ABB RobotStudio station: Solution_1.rspag

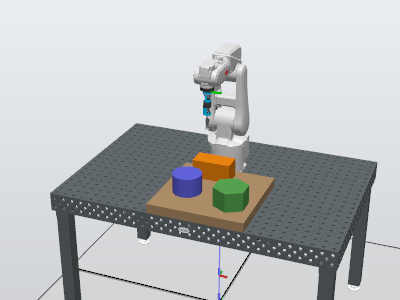
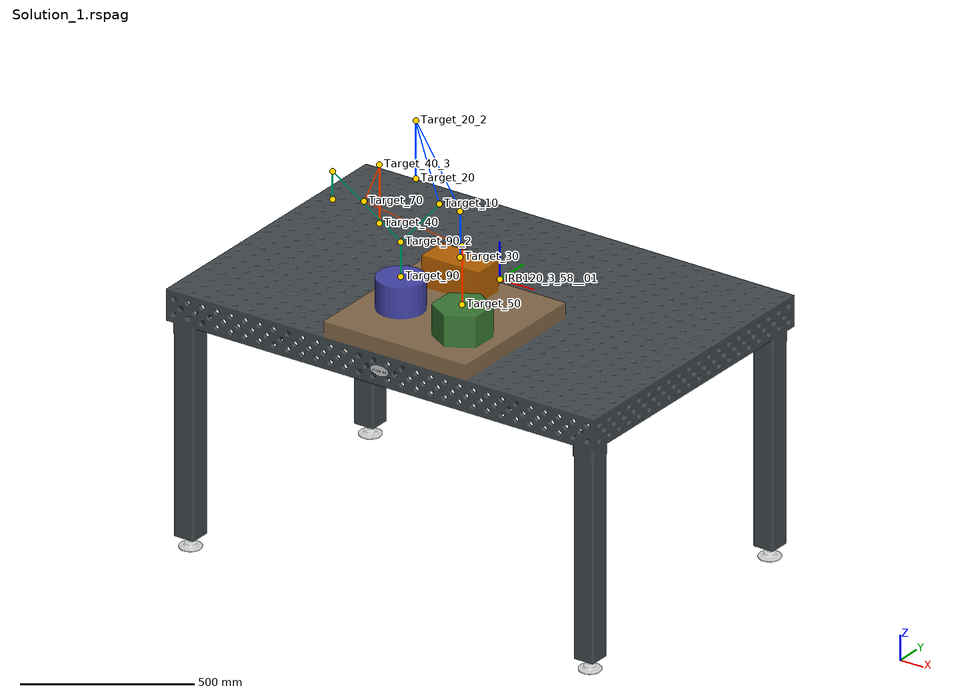
[picture v1: parts stored in the station drawn from their meshes, with robot base, taught points and paths (robot models come from the ABB library and are not in the file)]
--- station ---
Station Solution_1_Tutorial (saved by RobotStudio 22.3.10190.2)
Controller Controller1, task T_ROB1: task frame (RAPID world) sits at (0, 100, 830) mm, rotated rx 0 ry 0 rz -90 deg in the station
Controller Controller1
  mechanical unit ROB_1: IRB120_3_58__01, 6 joints, base frame (0, 0, 0) mm
Layout (positions relative to the parent item):
  - table [part] at (-200, -500, 830) mm, size 500 x 500 x 50 mm
  - object_1 [part] at (-200, -500, 830) mm, size 200 x 100 x 150 mm
  - object_2 [part] at (-200, -500, 830) mm, size 149.5 x 149.7 x 150 mm
  - object_3 [part] at (-200, -500, 830) mm, size 155.5 x 179.5 x 150 mm
  - siegmund_1500_1000 [part], size 1500 x 1010.3 x 830 mm
  - object_11 [part] at (-200, -500, 830) mm, size 200 x 100 x 150 mm
  - object_22 [part] at (-200, -500, 830) mm, size 149.5 x 149.7 x 150 mm
  - object_33 [part] at (-200, -500, 830) mm, size 155.5 x 179.5 x 150 mm
  - IRB120_3_58__01 [mechanism, from Robots\IRB120_3_58_G_01.rslib] at (0, 100, 830) mm, rotated rx 0 ry 0 rz -90 deg; joint values [0, 0, 0, 0, 1.5708, 0] (rad or m)
  - smc_gripper [mechanism, from Gripper_RS_tool\smc_gripper.rslib] at (0, -202, 1388) mm, rotated rx 180 ry 0 rz 90 deg
  - Attacher [smart component, from Components\Attacher.rslib]
      properties: Parent=smc_gripper; Flange=0; Child=object_1; Mount=false; Offset=[0 0 0]; Orientation=[0 0 0]
  - Detacher [smart component, from Components\Detacher.rslib]
      properties: Child=object_1; KeepPosition=true
  - Positioner [smart component, from Components\Positioner.rslib] at (-600, -150, 830) mm
      properties: Object=object_1; Position=[-0.6 -0.15 0.83]; Orientation=[0 0 0]; Reference=Global; ReferenceObject=(none)
  - Detacher_2 [smart component, from Components\Detacher.rslib]
      properties: Child=object_3; KeepPosition=true
  - Attacher_2 [smart component, from Components\Attacher.rslib]
      properties: Parent=smc_gripper; Flange=0; Child=object_3; Mount=false; Offset=[0 0 0]; Orientation=[0 0 0]
  - Attacher_3 [smart component, from Components\Attacher.rslib]
      properties: Parent=smc_gripper; Flange=0; Child=object_2; Mount=false; Offset=[0 0 0]; Orientation=[0 0 0]
  - Detacher_3 [smart component, from Components\Detacher.rslib]
      properties: Child=object_2; KeepPosition=true
  - Positioner_2 [smart component, from Components\Positioner.rslib]
      properties: Object=object_3; Position=[-0.7 -0.2 0.83]; Orientation=[0 0 0]; Reference=Global; ReferenceObject=(none)
  - Positioner_3 [smart component, from Components\Positioner.rslib]
      properties: Object=object_2; Position=[-0.65 -0.2 0.83]; Orientation=[0 0 0]; Reference=Global; ReferenceObject=(none)
  - Frame_1 [frame] at (0, 0, 197) mm
Attachment: smc_gripper is attached to IRB120_3_58__01 / Link6
Station signals: DI DI_TEST_01
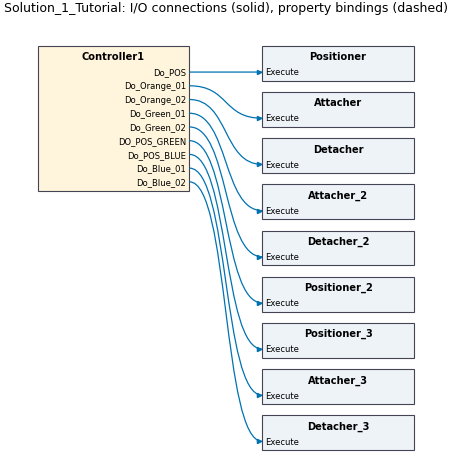
Station logic (signal -> signal, property => property):
  Controller1.Do_POS -> Positioner.Execute
  Controller1.Do_Orange_01 -> Attacher.Execute
  Controller1.Do_Orange_02 -> Detacher.Execute
  Controller1.Do_Green_01 -> Attacher_2.Execute
  Controller1.Do_Green_02 -> Detacher_2.Execute
  Controller1.DO_POS_GREEN -> Positioner_2.Execute
  Controller1.Do_POS_BLUE -> Positioner_3.Execute
  Controller1.Do_Blue_01 -> Attacher_3.Execute
  Controller1.Do_Blue_02 -> Detacher_3.Execute

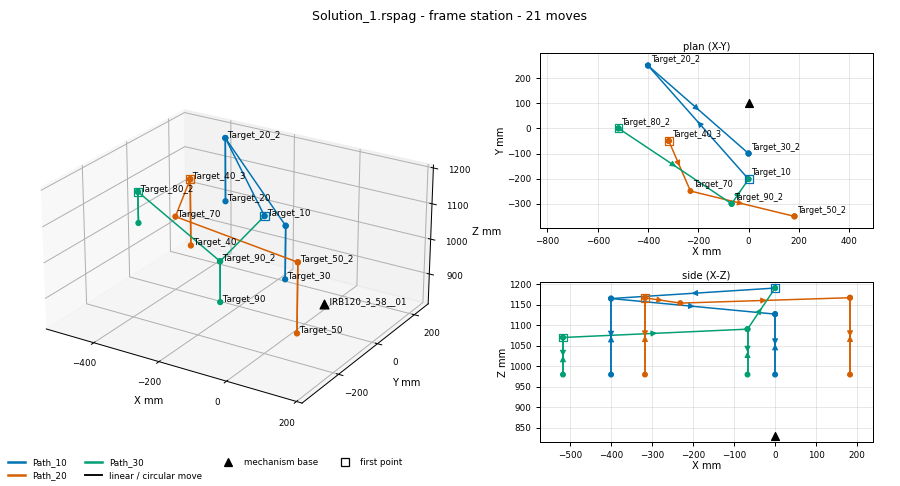
[picture p0: tool path of Solution_1.rspag in frame station, 21 of 21 moves have a stored position in this frame; points joined in program order, loops and branches not executed]
--- Backups/Controller1/RAPID/TASK1/PROGMOD/CalibData.mod ---
MODULE CalibData
    PERS tooldata smc_gripper:=[TRUE,[[0,0.004,197.001],[1,0,0,0]],[1,[0.207,-0.496,71.18],[1,0,0,0],0,0,0]];
ENDMODULE

--- Backups/Controller1/RAPID/TASK1/PROGMOD/Module1.mod ---
MODULE Module1

    CONST robtarget Target_10:=[[301.999956174,0.004,360.999],[-0.000000082,0,1,0],[0,0,0,0],[9E+09,9E+09,9E+09,9E+09,9E+09,9E+09]];
    CONST robtarget Target_20_2:=[[-150,-400,335.407930126],[-0.000000082,0,1,0],[-2,-1,-2,0],[9E+09,9E+09,9E+09,9E+09,9E+09,9E+09]];
    CONST robtarget Target_20:=[[-150,-400,150],[-0.000000082,0,1,0],[-2,-1,-2,0],[9E+09,9E+09,9E+09,9E+09,9E+09,9E+09]];
    CONST robtarget Target_30_2:=[[200,0,297.431267411],[-0.000000082,0,1,0],[-1,-1,-1,0],[9E+09,9E+09,9E+09,9E+09,9E+09,9E+09]];
    CONST robtarget Target_30:=[[200,0,150],[-0.000000082,0,1,0],[-1,-1,-1,0],[9E+09,9E+09,9E+09,9E+09,9E+09,9E+09]];
    CONST robtarget Target_40_3:=[[150,-317.298,337.140186548],[0,0.707106781,0.707106781,0],[-1,0,0,0],[9E+09,9E+09,9E+09,9E+09,9E+09,9E+09]];
    CONST robtarget Target_40:=[[150,-317.298,150],[0,0.707106781,0.707106781,0],[-1,0,0,0],[9E+09,9E+09,9E+09,9E+09,9E+09,9E+09]];
    CONST robtarget Target_50_2:=[[450,182.702,337.420142856],[0,0.707106781,0.707106781,0],[0,0,0,0],[9E+09,9E+09,9E+09,9E+09,9E+09,9E+09]];
    CONST robtarget Target_50:=[[450,182.702,150],[0,0.707106781,0.707106781,0],[0,0,1,0],[9E+09,9E+09,9E+09,9E+09,9E+09,9E+09]];
    CONST robtarget Target_70:=[[349.327498234,-231.175258404,324.28596128],[0,0.707106781,0.707106781,0],[0,0,0,0],[9E+09,9E+09,9E+09,9E+09,9E+09,9E+09]];
    CONST robtarget Target_80_2:=[[100,-517.298,240.437612888],[0,0.707106781,0.707106781,0],[0,0,0,0],[9E+09,9E+09,9E+09,9E+09,9E+09,9E+09]];
    CONST robtarget Target_80:=[[100,-517.298,150],[0,0.707106781,0.707106781,0],[0,0,0,0],[9E+09,9E+09,9E+09,9E+09,9E+09,9E+09]];
    CONST robtarget Target_90_2:=[[400,-67.298,260.778158702],[0,0.707106781,0.707106781,0],[0,0,0,0],[9E+09,9E+09,9E+09,9E+09,9E+09,9E+09]];
    CONST robtarget Target_90:=[[400,-67.298,150],[0,0.707106781,0.707106781,0],[0,0,0,0],[9E+09,9E+09,9E+09,9E+09,9E+09,9E+09]];
PROC main()
        PulseDO Do_POS; ! Dá to na nulu
        PulseDO DO_POS_GREEN;
        PulseDO Do_POS_BLUE;

        Path_20;
        Path_10;
        Path_30;


    ENDPROC
    PROC Path_10()
        MoveL Target_10,v300,z100,smc_gripper\WObj:=wobj0;
        MoveL Target_20_2,v300,z100,smc_gripper\WObj:=wobj0;
        MoveL Target_20,v300,fine,smc_gripper\WObj:=wobj0;

        WaitTime 0.25;
        ! DO ATTACH
        WaitTime 0.25;

        PulseDO Do_Orange_01;
        MoveL Target_20_2,v300,z100,smc_gripper\WObj:=wobj0;
        MoveL Target_30_2,v300,z100,smc_gripper\WObj:=wobj0;
        MoveL Target_30,v300,fine,smc_gripper\WObj:=wobj0;

        WaitTime 0.25;
        ! DO DETACH
        WaitTime 0.25;

        PulseDO Do_Orange_02;
        MoveL Target_30_2,v300,z100,smc_gripper\WObj:=wobj0;
    ENDPROC
    PROC Path_20()
        MoveL Target_40_3,v300,fine,smc_gripper\WObj:=wobj0;
        MoveL Target_40,v300,fine,smc_gripper\WObj:=wobj0;

        WaitTime 0.25;
        ! DO ATTACH
        WaitTime 0.25;

        PulseDO Do_Green_01;
        MoveL Target_40_3,v300,fine,smc_gripper\WObj:=wobj0;
        MoveL Target_70,v300,fine,smc_gripper\WObj:=wobj0;
        MoveL Target_50_2,v300,fine,smc_gripper\WObj:=wobj0;
        MoveL Target_50,v300,fine,smc_gripper\WObj:=wobj0;

        WaitTime 0.25;
        ! DO DETACH
        WaitTime 0.25;

        PulseDO Do_Green_02;
        MoveL Target_50_2,v300,fine,smc_gripper\WObj:=wobj0;
    ENDPROC
    PROC Path_30()
        MoveL Target_80_2,v300,z100,smc_gripper\WObj:=wobj0;
        MoveL Target_80,v300,fine,smc_gripper\WObj:=wobj0;

        WaitTime 0.25;
        ! DO ATTACH
        WaitTime 0.25;

        PulseDO Do_Blue_01;
        MoveL Target_80_2,v300,z100,smc_gripper\WObj:=wobj0;
        MoveL Target_90_2,v300,z100,smc_gripper\WObj:=wobj0;
        MoveL Target_90,v300,fine,smc_gripper\WObj:=wobj0;

        WaitTime 0.25;
        ! DO DETACH
        WaitTime 0.25;

        PulseDO Do_Blue_02;
        MoveL Target_90_2,v300,z100,smc_gripper\WObj:=wobj0;
        MoveL Target_10,v300,z100,smc_gripper\WObj:=wobj0;
    ENDPROC
ENDMODULE

--- Backups/Controller1/SYSPAR/EIO.cfg ---
EIO:CFG_1.0:6:1::
#
EIO_SIGNAL:

      -Name "Do_Orange_01" -SignalType "DO"

      -Name "Do_Orange_02" -SignalType "DO"

      -Name "Do_Attach" -SignalType "DO"

      -Name "Do_Detach" -SignalType "DO"

      -Name "Do_POS" -SignalType "DO"

      -Name "Do_Green_01" -SignalType "DO"

      -Name "Do_Green_02" -SignalType "DO"

      -Name "DO_POS_GREEN" -SignalType "DO"

      -Name "Do_POS_BLUE" -SignalType "DO"

      -Name "Do_Blue_01" -SignalType "DO"

      -Name "Do_Blue_02" -SignalType "DO"
